Staubli VAL3: Message.pgx

program Message(string x_sMsg, bool x_bLogShow)
  local num l_ni
begin
  //显示操作信息
  //x_sMsg:需要显示的信息
  //x_bLogShow:
  //--true:在userpage和log同时显示；
  //--false:仅在userpage中显示

  for l_ni=0 to 7
    if sMsg[l_ni]==""
      sMsg[l_ni]=x_sMsg
      l_ni=8
    elseIf l_ni==7
      for l_ni=0 to 6
        sMsg[l_ni]=sMsg[l_ni+1]
      endFor
      sMsg[l_ni]=x_sMsg
    endIf
  endFor

  for l_ni=0 to 7
    gotoxy(1,3+l_ni)
    put(sMsg[l_ni]+"     ")
  endFor
  //
  if x_bLogShow
    logMsg(sMsg)
  endIf
end
